ABB RAPID module: wenglorUserConfig.modx

MODULE wenglorUserConfig
    !***********************************************************
    !
    ! Module:  wenglorUserConfig
    !
    ! Author: wenglor sensoric GmbH
    !
    ! Version: 1.3.0
    !
    ! Description:
    !   This module contains global variables and helper functions.
    !
    ! How to start:
    ! * Set the port and IP address in the section below, as well as the use case "camera_on_robot" or "camera_not_on_robot".
    ! * Check whether ABB is selected in the robot manufacturer drop-down of the robot server on the machine vision device website (e.g. B60, MVC).
    ! * Run calibration if it has not been done yet.
    !
    ! How to do the calibration:
    ! * Rename the uniVision calibration job in the section below so it matches your selected name.
    ! * Set at least five calibration poses. The variance of the calibration movements matters, not the variance of the calibration poses.
    ! * Please use the calibration pose variables from the section below wCalibPose1, wCalibPose2, ...
    ! * If you want to use more than 5 calibration poses, follow the naming scheme and extend the calibration pose sequence in wenglorCalibration - runCalibration().
    ! * Check if the movements are safe by moving manually from pose to pose in debug mode.
    ! * Name the calibration target you are using in the constant W_CALIBRATION_TARGET in the section below.
    ! * If your camera is not mounted on the robot, also set a wDetectionPose pose, as the calibration target will be placed
    !   on the object ground in the second step of calibration in this case.
    !   The robot will move to the detection pose to detect the calibration target placed on the object ground.
    !
    ! After the calibration:
    ! * Take a look at the main procedure of wenglorDetect.
    ! * Replace the wDetectionPose pose with the one you are using.
    ! * Ensure your tool is properly set.
    ! * If you notice a height offset, check whether the uniVision job is set properly, especially the height offset from the calibration target to
    !   the object in the "Device Robot Vision".
    ! * This is just a basic example. If you want to handle multiple objects with just one wDetectionPose,
    !   use different shape models, the additional values you linked in uniVision, or access an object pose via an index.
    !   check the uniVision operating instructions DNNF023.
    !
    !***********************************************************

    !*********************************************************** USER CONFIG ********************************************************!
    ! Replace IP address and port with your setup.
    CONST string W_VISION_DEVICE_IP:="192.168.100.1";
    CONST num W_VISION_DEVICE_PORT:=32006;

    ! Comment out the correct line depending on the selected camera/robot setup
    CONST string W_USE_CASE:="camera_on_robot";
    !CONST string W_USE_CASE := "camera_not_on_robot";

    ! Replace with the calibration target you are using
	! Calibration target:
	! "zvzj001" | "zvzj002" | "zvzj003" | "zvzj004" |
	! "24x30mm" | "375x550mm" | "550x800mm"
    ! if you are using zvzj005, replace with zvzj001 and
    ! if you are using zvzj006, replace with zvzj002
    CONST string W_CALIBRATION_TARGET:="zvzj001";
    ! Replace the calibration job with the one you created in uniVision
    CONST string W_CALIBRATION_JOB:="calibration.u3p";
    CONST string W_DETECT_OBJECTS_JOB:="find_objects.u3p";
    CONST string W_DETECT_TARGET_JOB:="find_target.u3p";

    CONST string W_USER_COMMAND:="singleDetection";
    !CONST string W_USER_COMMAND:="multiDetection";
    !CONST string W_USER_COMMAND:="updateReferenceFrame";


    ! Adjust validation z safety offset [mm]
    CONST num W_SAFETY_OFFSET_MM:=10;

    ! Set speed for calibration movements here
    CONST speeddata W_CALIB_SPEED:=v100;
    ! Set calibration poses here
    VAR robtarget wCalibPose1:=[[0,0,0],[0,0,0,0],[0,0,0,0],[0,0,0,0,0,0]];
    VAR robtarget wCalibPose2:=[[0,0,0],[0,0,0,0],[0,0,0,0],[0,0,0,0,0,0]];
    VAR robtarget wCalibPose3:=[[0,0,0],[0,0,0,0],[0,0,0,0],[0,0,0,0,0,0]];
    VAR robtarget wCalibPose4:=[[0,0,0],[0,0,0,0],[0,0,0,0],[0,0,0,0,0,0]];
    VAR robtarget wCalibPose5:=[[0,0,0],[0,0,0,0],[0,0,0,0],[0,0,0,0,0,0]];

    ! Set wDetectionPose here for the "camera_not_on_robot" case.
    ! Otherwise, do not change it, as it will be updated in runCalibration().
    PERS robtarget wDetectionPose:=[[0,0,0],[0,0,0,0],[0,0,0,0],[0,0,0,0,0,0]];


    !*********************** Mobile Platform use case *********************************

    ! Set to TRUE if you have taught the poses inside the machine. Otherwise, the program will stop after updating the reference frame (wReferenceFrame),
    ! so you can approach the machine and teach the poses relative to the wReferenceFrame
    CONST bool W_MACHINE_POSES_TAUGHT := FALSE;

    ! This is the reference frame for all fixed poses inside the machine
    PERS wobjdata wReferenceFrame:=[FALSE,TRUE,"",[[0,0,0],[1,0,0,0]],[[0,0,0],[1,0,0,0]]];

    ! This is one dummy pose that represents any pose in the machine relative to the wReferenceFrame
    PERS robtarget wPoseInMachine:=[[0,0,0],[0,0,0,0],[0,0,0,0],[0,0,0,0,0,0]];

    !******************************************************* END USER CONFIG ********************************************************!

ENDMODULE
